FUNCTION_BLOCK TcSynchronizedAxisCommand IMPLEMENTS itfSynchronizedAxisCommand
VAR_INPUT
END_VAR
VAR_OUTPUT
END_VAR
VAR
END_VAR

{warning 'add method implementation '}
METHOD Abort : MC_Error
END_METHOD

{warning 'add property implementation'}
PROPERTY Active : BOOL
GET
END_GET
END_PROPERTY

{warning 'add property implementation'}
PROPERTY Busy : BOOL
GET
END_GET
END_PROPERTY

{warning 'add property implementation'}
PROPERTY Command : MC_COMMAND_REF
GET
END_GET
END_PROPERTY

{warning 'add property implementation'}
PROPERTY CommandAborted : BOOL
GET
END_GET
END_PROPERTY

{warning 'add property implementation'}
PROPERTY Done : BOOL
GET
END_GET
END_PROPERTY

{warning 'add property implementation'}
PROPERTY Error : BOOL
GET
END_GET
END_PROPERTY

{warning 'add property implementation'}
PROPERTY ErrorId : MC_Error
GET
END_GET
END_PROPERTY

{warning 'add property implementation'}
PROPERTY InSync : BOOL
GET
Insync:= Geared;
END_GET
END_PROPERTY

{warning 'add method implementation '}
METHOD Update 		: MC_Error
VAR_INPUT
	Position		: REAL;
	Velocity		: REAL;
	EndVelocity		: REAL;
	Acceleration	: REAL;
	Deceleration	: REAL;
	Jerk			: REAL;
END_VAR
END_METHOD

{warning 'add method implementation '}
METHOD Wait 		: MC_Error (* This method only makes sense in the IEC 61499 environment*)
VAR_INPUT
	Timeout			: TIME;
	AbortOnTimeout	: BOOL;
END_VAR
END_METHOD

END_FUNCTION_BLOCK

(* stored: Version 1.1.0.1, ProductVersion 3.1.4024.12
   POU TcSynchronizedAxisCommand: Id {dee37af4-cc16-4c69-b646-3f672cb97306}, SpecialFunc None
   Method Abort: Id {32420f3d-fe16-45ed-96a2-fe0f4af2554c}
   Property Active: Id {405139b7-1924-4787-af06-3f6761fc23bc}
   Get Get: Id {4da5366b-02e2-4bdf-9651-c048c4c27c73}
   Property Busy: Id {06741541-e49c-43bb-8ef6-5a50bca72f39}
   Get Get: Id {b61d6362-c193-4776-9ddb-d38d5017c8e3}
   Property Command: Id {ce54ca8b-e3b1-47a5-b2e6-aa375c6e81f7}
   Get Get: Id {8eb99693-14f4-4771-8504-0d5cd1f308f1}
   Property CommandAborted: Id {4158dd63-11c0-4f55-815a-c72388bc3391}
   Get Get: Id {17442d6c-2014-4562-a13a-4b9bc0264318}
   Property Done: Id {e10a6386-a699-4579-81a3-ac6e43307d1b}
   Get Get: Id {22c20995-eaf9-47da-8e7a-d52b1f3f407f}
   Property Error: Id {29b8fe53-9c4c-45c9-8cc8-9362f783cb46}
   Get Get: Id {013e13c3-866b-4d35-935e-5a97ebe88978}
   Property ErrorId: Id {3fc97fc9-3580-4d4f-8d19-b26cfa2ae1e5}
   Get Get: Id {ca7353a9-24b7-47d3-a2eb-fbe515c6f6b3}
   Property InSync: Id {78392d25-2d35-4e46-ae17-8b8661ec2c4e}
   Get Get: Id {1a3865a3-e28a-4655-a0b1-217c6d132d7d}
   Method Update: Id {63972c03-57b5-46cc-95e9-e5c4537e4641}
   Method Wait: Id {8fa71d3f-a921-4d37-93eb-050f25575da9} *)
